# EPICS substitutions: snmpApp/Db/ups.substitutions
file "toshibaUPSsnmp.template"
{
  pattern { Sys, Dev , IP, C}
 { "XF:23ID-CT", "{UPS:1}", "10.23.3.1", "public" }
#  { "XF:23ID-CT", "{UPS:2}", "10.23.3.2", "public" }
}
